(* IEC 61131-3 sources: generating_plc_code_with_llms/Code#2/ChatGPT_4/second run, 21 files *)

(* ---- 14.st ---- *)
// 34.95s
// 4
FUNCTION FC1001 : BOOL
VAR_INPUT
    MEW: REAL;  (* Measured value from the sensor *)
    SP: REAL;   (* Setpoint value *)
    HYS: REAL;  (* Hysteresis percentage *)
END_VAR
VAR_IN_OUT
    OUT: BOOL;  (* Output to be controlled *)
END_VAR
VAR
    P_HYS: REAL;  (* Absolute hysteresis value *)
END_VAR

P_HYS := SP * HYS / 100.0;  (* Calculate the hysteresis value *)

IF MEW > (SP + P_HYS) THEN
    OUT := TRUE;  (* Turn on output if measured value exceeds SP + hysteresis *)
ELSIF MEW < (SP - P_HYS) THEN
    OUT := FALSE;  (* Turn off output if measured value falls below SP - hysteresis *)
END_IF;

FC1001 := OUT;  (* Return the current state of the output *)

END_FUNCTION

(* ---- 15.st ---- *)
// 64.56s
// 4
FUNCTION FC1002 : BOOL
VAR_INPUT
    E_A : BOOL;     (* Switch for enabling/disabling the monitoring system *)
    SENSOR : BOOL;  (* Ultrasonic sensor input *)
    ZEITW : TIME;   (* Time duration for switching from warning to alarm *)
END_VAR
VAR_IN_OUT
    ZEIT : TON;     (* Timer for measuring the duration of perception *)
    P_HU : BOOL;    (* Horn for acoustic warning signal *)
    P_AL : BOOL;    (* Alarm signal *)
END_VAR

(* Monitoring system activation *)
IF E_A THEN
    (* When monitoring system is enabled *)
    IF SENSOR THEN
        ZEIT(IN := TRUE, PT := ZEITW);
        IF ZEIT.Q THEN
            P_HU := FALSE;  (* Turn off horn after time window *)
            P_AL := TRUE;   (* Activate alarm *)
        ELSE
            P_HU := TRUE;   (* Activate horn if object/person is detected *)
        END_IF;
    ELSE
        ZEIT(IN := FALSE);
        P_HU := FALSE;  (* Turn off horn if no object/person is detected *)
    END_IF;
ELSE
    (* When monitoring system is disabled *)
    P_HU := FALSE;
    P_AL := FALSE;
    ZEIT(IN := FALSE);
END_IF;

FC1002 := E_A;  (* Return the status of the monitoring system *)

END_FUNCTION

(* ---- 18.st ---- *)
// 37.69s
// 4
FUNCTION FC1003 : VOID
VAR_INPUT
    IN_R : REAL;      (* Input real value *)
    IN_MAX : REAL;    (* Input range maximum *)
    IN_MIN : REAL;    (* Input range minimum *)
    OUT_MAX : REAL;   (* Output range maximum *)
    OUT_MIN : REAL;   (* Output range minimum *)
END_VAR
VAR_OUTPUT
    OUT_R : REAL;     (* Output real value *)
    FEH : BOOL;       (* Error flag in case of invalid range *)
END_VAR
VAR_TEMP
    DIFF1 : REAL;     (* Temporary variable for differences *)
    DIFF2 : REAL;     (* Temporary variable for differences *)
END_VAR

(* Check for valid input range to avoid division by zero *)
IF IN_MAX <= IN_MIN THEN
    FEH := TRUE;
    RETURN;
END_IF;

(* Calculate the differences *)
DIFF1 := IN_MAX - IN_MIN;
DIFF2 := OUT_MAX - OUT_MIN;

(* Map the input value to the output range *)
OUT_R := OUT_MIN + ((IN_R - IN_MIN) * DIFF2) / DIFF1;

(* Set the error flag to false as no error occurred *)
FEH := FALSE;

END_FUNCTION

(* ---- 19.st ---- *)
// 43.16s
// 4
FUNCTION_BLOCK FB1005
VAR_INPUT
    START : BOOL;    (* Signal to start and end measurement *)
    DICKE : REAL;    (* Thickness measurement from lasers *)
    V_MAX : REAL;    (* Maximum tolerance value for thickness *)
    V_MIN : REAL;    (* Minimum tolerance value for thickness *)
END_VAR
VAR_OUTPUT
    D_MAX : REAL;    (* Maximum measured thickness *)
    D_MIN : REAL;    (* Minimum measured thickness *)
    P1 : BOOL;       (* Reject light indicator *)
END_VAR
VAR
    FO : BOOL;       (* Flag to indicate ongoing measurement *)
END_VAR

IF START THEN
    IF NOT FO THEN
        (* Start of a new measurement *)
        FO := TRUE;
        D_MAX := DICKE;
        D_MIN := DICKE;
    ELSE
        (* Ongoing measurement *)
        IF DICKE > D_MAX THEN
            D_MAX := DICKE;
        END_IF;

        IF DICKE < D_MIN THEN
            D_MIN := DICKE;
        END_IF;
    END_IF;
ELSE
    IF FO THEN
        (* End of measurement *)
        FO := FALSE;

        (* Check if measured values are outside tolerance range *)
        IF D_MAX > V_MAX OR D_MIN < V_MIN THEN
            P1 := TRUE;  (* Set reject light *)
        ELSE
            P1 := FALSE; (* Reset reject light *)
        END_IF;
    END_IF;
END_IF;

END_FUNCTION_BLOCK

(* ---- 20.st ---- *)
// 32.83s
// 3
FUNCTION_BLOCK INTERLOCK
VAR_INPUT
    I1 : BOOL;  (* Input for controlling Q1 *)
    I2 : BOOL;  (* Input for controlling Q2 *)
    TL : TIME;  (* Dead time between switching outputs *)
END_VAR
VAR_OUTPUT
    Q1 : BOOL;  (* Output Q1 *)
    Q2 : BOOL;  (* Output Q2 *)
END_VAR
VAR
    T1 : TOF;  (* Off-delay timer for Q1 *)
    T2 : TOF;  (* Off-delay timer for Q2 *)
END_VAR

(* Timer logic for Q1 *)
T1(IN := NOT Q1, PT := TL);
IF I1 AND T2.Q THEN
    Q1 := TRUE;
    Q2 := FALSE;
END_IF;

(* Timer logic for Q2 *)
T2(IN := NOT Q2, PT := TL);
IF I2 AND T1.Q THEN
    Q2 := TRUE;
    Q1 := FALSE;
END_IF;

END_FUNCTION_BLOCK

(* ---- 21.st ---- *)
// 144.85s
// weiter generieren
// 2
FUNCTION_BLOCK BURNER
VAR_INPUT
    IN : BOOL;
    STAGE2 : BOOL;
    OVER_TEMP : BOOL;
    OIL_TEMP : BOOL := TRUE;
    FLAME : BOOL;
    RST : BOOL;
    RST_TIMER : BOOL;
    PRE_HEAT_TIME : TIME := t#5s;
    PRE_VENT_TIME : TIME := t#15s;
    PRE_IGNITE_TIME : TIME := t#15s;
    POST_IGNITE_TIME : TIME := t#25s;
    STAGE2_DELAY : TIME := t#10s;
    SAFETY_TIME : TIME := t#5s;
    LOCKOUT_TIME : TIME := t#10s;
    MULTIPLE_IGNITION : BOOL := TRUE;
    KW1 : REAL;
    KW2 : REAL;
END_VAR
VAR_OUTPUT
    MOTOR : BOOL;
    COIL1 : BOOL;
    COIL2 : BOOL;
    PRE_HEAT : BOOL;
    IGNITE : BOOL;
    FAIL : BOOL;
    KWH : REAL;
    STATUS : BYTE;
END_VAR
VAR_IN_OUT
    RUNTIME1 : UDINT;
    RUNTIME2 : UDINT;
    CYCLES : UDINT;
END_VAR
VAR
    state : INT := 0;  (* Operational state of the burner *)
    last : TIME;  (* Last time an operation started *)
    tx : TIME;  (* Transition time for next state *)
    last_change : TIME;  (* Last time state changed *)
    timer1 : TON;  (* Timer for various operational delays *)
    timer2 : TON;  (* Timer for lockout period *)
    oil_temp_last : BOOL := FALSE;  (* Last state of OIL_TEMP *)
    cycles2 : UDINT;  (* Cycle count for stage 2 *)
END_VAR

(* Reset functionality *)
IF RST THEN
    state := 0;
    FAIL := FALSE;
    STATUS := 110;  (* Wait for Start signal *)
    timer2(IN := FALSE);  (* Reset lockout timer *)
    MOTOR := FALSE;
    PRE_HEAT := FALSE;
    IGNITE := FALSE;
    COIL1 := FALSE;
    COIL2 := FALSE;
    RETURN;
END_IF;

(* Lockout timer check *)
timer2(IN := RST_TIMER, PT := LOCKOUT_TIME);
IF timer2.Q THEN
    RST_TIMER := FALSE;  (* Reset RST_TIMER after lockout period *)
END_IF;

(* Main state machine for burner operation *)
CASE state OF
    0:
        IF IN AND NOT OVER_TEMP AND NOT timer2.Q THEN
            state := 1;
            PRE_HEAT := TRUE;
            last_change := tx;
            timer1(IN := TRUE, PT := PRE_HEAT_TIME);
        END_IF;
    1:
        IF timer1.Q THEN
            IF NOT OIL_TEMP THEN
                FAIL := TRUE;
                STATUS := 1;  (* Fuel oil warming has not responded within PRE_HEAT_TIME *)
                state := 9;  (* Error state *)
            ELSE
                state := 2;  (* Proceed to next stage *)
                MOTOR := TRUE;
                last_change := tx;
                timer1(IN := TRUE, PT := PRE_VENT_TIME);  (* Start ventilation period *)
            END_IF;
        END_IF;
    2:
        IF timer1.Q THEN
            state := 3;
            IGNITE := TRUE;
            last_change := tx;
            timer1(IN := TRUE, PT := PRE_IGNITE_TIME + SAFETY_TIME);  (* Ignition and safety period *)
        END_IF;
    3:
        IF FLAME THEN
            state := 4;
            COIL1 := TRUE;  (* Burner running on stage 1 *)
            STATUS := 112;
            last_change := tx;
            RUNTIME1 := RUNTIME1 + 1;
            IF STAGE2 THEN
                timer1(IN := TRUE, PT := STAGE2_DELAY);  (* Delay for stage 2 activation *)
            END_IF;
        ELSIF timer1.Q THEN
            FAIL := TRUE;
            STATUS := 4;  (* Safety time was passed without a flame *)
            state := 9;  (* Error state *)
        END_IF;
    4:
        IF timer1.Q AND STAGE2 THEN
            state := 5;
            COIL2 := TRUE;  (* Burner running on stage 2 *)
            STATUS := 113;
            RUNTIME2 := RUNTIME2 + 1;
        END_IF;
    9:
        MOTOR := FALSE;
        PRE_HEAT := FALSE;
        IGNITE := FALSE;
        COIL1 := FALSE;
        COIL2 := FALSE;
        RST_TIMER := TRUE;  (* Start lockout timer *)
        state := 0;  (* Reset state after handling error *)
END_CASE;

(* Handle OVER_TEMP condition *)
IF OVER_TEMP THEN
    FAIL := TRUE;
    STATUS := 9;  (* Boiler overheating contact has tripped *)
    MOTOR := FALSE;
    PRE_HEAT := FALSE;
    IGNITE := FALSE;
    COIL1 := FALSE;
    COIL2 := FALSE;
    state := 9;  (* Set error state *)
END_IF;

END_FUNCTION_BLOCK

(* ---- 1.st ---- *)
// 18.4s
// 4
VAR
    xAllOn : BOOL;
    xAllOff : BOOL;
    xAlarm1 : BOOL;
    xAlarm2 : BOOL;
END_VAR

IF xAllOn THEN
    xAlarm1 := TRUE;
    xAlarm2 := TRUE;
    xAllOn := FALSE;
END_IF;

IF xAllOff THEN
    xAlarm1 := FALSE;
    xAlarm2 := FALSE;
    xAllOff := FALSE;
END_IF;

(* ---- 10.st ---- *)
// 16.0s
// 4
VAR_INPUT
    X : REAL;
END_VAR

VAR
    SigmoidResult : REAL;
END_VAR

SigmoidResult := 1 / (1 + EXP(-X));

(* ---- 11.st ---- *)
// 17.44s
// 4
VAR_INPUT
    x : REAL;  (* Input number *)
END_VAR

VAR
    signResult : INT;  (* Result of the sign function *)
END_VAR

IF x > 0 THEN
    signResult := 1;  (* Positive number *)
ELSIF x < 0 THEN
    signResult := -1;  (* Negative number *)
ELSE
    signResult := 0;  (* Zero *)
END_IF;

(* ---- 12.st ---- *)
// 13.41s
// 4
VAR
    X : REAL;         (* Input for the hyperbolic sine function *)
    SinhResult : REAL; (* Result of sinh(x) *)
END_VAR

SinhResult := (EXP(X) - EXP(-X)) / 2;

(* ---- 13.st ---- *)
// 20.21s
// 2
VAR CONSTANT
    MAXNUMBERS : UINT := 99;  (* The upper index of the array *)
END_VAR

VAR
    aNumbers : ARRAY[0..MAXNUMBERS] OF INT;  (* Array of 100 random numbers *)
    nCnt : INT;                              (* Counter for the loop *)
END_VAR

nCnt := 0;

REPEAT
    IF aNumbers[nCnt] = 10 THEN
        EXIT;  (* Exit the loop if the number 10 is found *)
    END_IF;

    nCnt := nCnt + 1;
UNTIL nCnt > MAXNUMBERS;  (* Continue until the end of the array is reached *)

(* ---- 16.st ---- *)
// 57.71s
// 4
VAR
    North_green : BOOL;
    North_yellow : BOOL;
    North_red : BOOL;
    East_green : BOOL;
    East_yellow : BOOL;
    East_red : BOOL;
    T1 : TON;
END_VAR

(* Start the timer *)
T1(IN := TRUE, PT := T#10000MS);

(* Control the North and East traffic lights based on the elapsed time of the timer *)
IF T1.ET < T#5000MS THEN
    (* 0ms to 5000ms: North green, East red *)
    North_green := TRUE;
    North_yellow := FALSE;
    North_red := FALSE;
    East_green := FALSE;
    East_yellow := FALSE;
    East_red := TRUE;
ELSIF T1.ET < T#5500MS THEN
    (* 5000ms to 5500ms: North yellow, East red *)
    North_green := FALSE;
    North_yellow := TRUE;
    North_red := FALSE;
    East_green := FALSE;
    East_yellow := FALSE;
    East_red := TRUE;
ELSIF T1.ET < T#9500MS THEN
    (* 5500ms to 9500ms: North red, East green *)
    North_green := FALSE;
    North_yellow := FALSE;
    North_red := TRUE;
    East_green := TRUE;
    East_yellow := FALSE;
    East_red := FALSE;
ELSE
    (* 9500ms to 10000ms: North red, East yellow *)
    North_green := FALSE;
    North_yellow := FALSE;
    North_red := TRUE;
    East_green := FALSE;
    East_yellow := TRUE;
    East_red := FALSE;
END_IF;

(* Reset the timer at the end of the cycle *)
IF T1.Q THEN
    T1.IN := FALSE;
    T1(IN := TRUE);  (* Restart the timer *)
END_IF;

(* ---- 17.st ---- *)
// 28.0s
// 3
VAR
    aiOutside : INT;       (* Analog input for outside temperature *)
    aiHumidity : INT;      (* Analog input for humidity *)
    sShowText : STRING[80];(* String to display the message *)
END_VAR

(* Convert the analog inputs to temperature and humidity values *)
(* Assuming the range of the analog input is from 0 to 32767 and this corresponds to -40 to 60 °C for temperature and 0 to 100% for humidity *)
VAR
    fTemperature : REAL; (* Temperature in degrees Celsius *)
    fHumidity : REAL;    (* Humidity in percentage *)
END_VAR

fTemperature := (aiOutside / 32767.0) * 100.0 - 40.0;  (* Conversion formula *)
fHumidity := (aiHumidity / 32767.0) * 100.0;           (* Conversion formula *)

(* Evaluate temperature and humidity to set the display text *)
IF fTemperature < 18 THEN
    sShowText := 'Cold';
ELSIF fTemperature <= 25 THEN
    IF fHumidity >= 40 AND fHumidity <= 75 THEN
        sShowText := 'Opt';
    ELSE
        sShowText := 'Temp. OK';
    END_IF;
ELSE
    sShowText := 'Hot';
END_IF;

(* ---- 2.st ---- *)
// 26.75s
// 4
VAR_INPUT
    N : INT;
    K : INT;
END_VAR

VAR
    Result : LREAL;  (* Using LREAL for potentially large results *)
    i : INT;
END_VAR

(* Initialize result *)
Result := 1;

(* Adjust K for optimization *)
IF K > N - K THEN
    K := N - K;
END_IF;

(* Calculate binomial coefficient *)
FOR i := 0 TO K - 1 DO
    Result := Result * (N - i) / (i + 1);
END_FOR;

(* ---- 3.st ---- *)
// 17.02s
// 3
VAR_INPUT
    X : INT;
END_VAR

VAR
    t1 : DINT := 0;
    t2 : DINT := 1;
    nextTerm : DINT := 0;
    i : INT;
END_VAR

IF X = 0 THEN
    nextTerm := 0;
ELSIF X = 1 THEN
    nextTerm := 1;
ELSE
    FOR i := 2 TO X DO
        nextTerm := t1 + t2;
        t1 := t2;
        t2 := nextTerm;
    END_FOR;
END_IF;

(* ---- 4.st ---- *)
// 26.41s
// 2
VAR
    aiLevel : INT;           (* Analog input representing the fill level *)
    PercentLevel : UINT;     (* Fill level as a percentage *)
    doLow : BOOL;            (* Output for low level indication *)
    doOk : BOOL;             (* Output for ok level indication *)
    doHigh : BOOL;           (* Output for high level indication *)
    doAlarm : BOOL;          (* Output for alarm indication *)
END_VAR

(* Convert the analog input to a percentage *)
PercentLevel := UINT(aiLevel * 100 / 32767);

(* Check the level and set outputs accordingly *)
CASE PercentLevel OF
    0..1:
        BEGIN
            doLow := TRUE;
            doOk := FALSE;
            doHigh := FALSE;
            doAlarm := TRUE; (* Activate alarm for less than 1% *)
        END
    2..79:
        BEGIN
            doLow := FALSE;
            doOk := TRUE;
            doHigh := FALSE;
            doAlarm := FALSE;
        END
    80..100:
        BEGIN
            doLow := FALSE;
            doOk := FALSE;
            doHigh := TRUE;
            doAlarm := FALSE;
        END
END_CASE;

(* ---- 5.st ---- *)
// 50.7s
// 4
VAR
    Start_Loop : BOOL := FALSE;
    one_hour : TIME := T#1h;            (* 1 hour duration for timer *)
    One_Hour_Timer : TON;               (* Timer for 1 hour countdown *)
    Gate_Open : BOOL := FALSE;          (* Indicates if gate is open *)
    Close_Gate_Inst : BOOL := FALSE;    (* Instruction to close gate *)
    Sensed_Car : BOOL := FALSE;         (* Detects presence of car *)
    Sensed_Car_Inst : BOOL := FALSE;    (* Car detection instance *)
    Sensed_App : BOOL := FALSE;         (* Detects signal from app *)
    Mobile_Inst : BOOL := FALSE;        (* Mobile app detection instance *)
    Auth : STRING;                      (* Authentication string *)
    my_defined_str : STRING := 'abcd';  (* Defined authentication string *)
END_VAR

(* Timer control *)
IF Start_Loop = FALSE THEN
    One_Hour_Timer(IN := TRUE, PT := one_hour);
ELSE
    One_Hour_Timer(IN := FALSE);
END_IF;

(* Check if timer has timed out and gate is open *)
IF One_Hour_Timer.Q AND Gate_Open THEN
    Close_Gate_Inst := TRUE;
    Gate_Open := FALSE;
END_IF;

(* Check for car or app presence and correct authentication *)
IF (Sensed_Car OR Sensed_App) AND (Auth = my_defined_str) THEN
    Gate_Open := TRUE;
    Sensed_Car_Inst := Sensed_Car;
    Mobile_Inst := Sensed_App;
ELSE
    IF NOT One_Hour_Timer.Q THEN
        Close_Gate_Inst := FALSE;
    END_IF;
END_IF;

(* ---- 6.st ---- *)
// 47.53s
// 3
VAR CONSTANT
    WAIT : UINT := 0;
    TOP_POSITION : UINT := 1;
    BOTTOM_POSITION : UINT := 2;
    GETBOX : UINT := 3;
    UNLOAD_POSITION : UINT := 4;
    UNLOAD_BOX : UINT := 5;
END_VAR

VAR
    (* digital outputs *)
    doConvTop : BOOL;
    doConvBottom : BOOL;
    doConvLift : BOOL;
    doLiftTop : BOOL;
    doLiftBottom : BOOL;
    doLiftUnload : BOOL;
    (* digital inputs *)
    diConvTop : BOOL;
    diConvBottom : BOOL;
    diLiftTop : BOOL;
    diLiftBottom : BOOL;
    diLiftUnload : BOOL;
    diBoxLift : BOOL;
    (* status variables *)
    selectLift : UINT;
    ConvTopOn : BOOL;
    ConvBottomOn : BOOL;
END_VAR

(* Handle the conveyor belts *)
IF diConvTop THEN
    doConvTop := FALSE;
    selectLift := TOP_POSITION;
END_IF;

IF diConvBottom THEN
    doConvBottom := FALSE;
    selectLift := BOTTOM_POSITION;
END_IF;

(* Control the lift *)
CASE selectLift OF
    TOP_POSITION:
        IF NOT diLiftTop THEN
            doLiftTop := TRUE;
            doLiftBottom := FALSE;
            doLiftUnload := FALSE;
        ELSIF diLiftTop THEN
            doConvLift := TRUE;
            IF diBoxLift THEN
                selectLift := UNLOAD_POSITION;
            END_IF;
        END_IF;

    BOTTOM_POSITION:
        IF NOT diLiftBottom THEN
            doLiftBottom := TRUE;
            doLiftTop := FALSE;
            doLiftUnload := FALSE;
        ELSIF diLiftBottom THEN
            doConvLift := TRUE;
            IF diBoxLift THEN
                selectLift := UNLOAD_POSITION;
            END_IF;
        END_IF;

    UNLOAD_POSITION:
        doConvLift := FALSE;
        doLiftUnload := TRUE;
        IF diLiftUnload THEN
            selectLift := UNLOAD_BOX;
        END_IF;

    UNLOAD_BOX:
        doLiftUnload := FALSE;
        IF NOT diBoxLift THEN
            selectLift := WAIT;
        END_IF;

    WAIT:
        doLiftTop := FALSE;
        doLiftBottom := FALSE;
        doLiftUnload := FALSE;
END_CASE;

(* ---- 7.st ---- *)
// 18.24s
// 2
VAR CONSTANT
    MAX_INDEX: USINT := 4;  (* Represents the highest index for load receptors *)
END_VAR

VAR
    aWeights : ARRAY[0..MAX_INDEX] OF INT;  (* Array of load values from receptors *)
    iCnt : USINT;                           (* Loop counter *)
    sumWeight : DINT;                       (* Total sum of weights *)
    avgWeight : INT;                        (* Average weight *)
END_VAR

(* Initialize sum *)
sumWeight := 0;

(* Calculate the sum of the weights *)
FOR iCnt := 0 TO MAX_INDEX DO
    sumWeight := sumWeight + aWeights[iCnt];
END_FOR;

(* Calculate the average weight, dividing by the number of receptors *)
avgWeight := sumWeight / (MAX_INDEX + 1);

(* ---- 8.st ---- *)
// 29.25s
// 3
VAR_INPUT
    X : REAL;  (* Input for the Lambert W function *)
END_VAR

VAR
    w : REAL;      (* Approximation of W(x) *)
    i : INT;       (* Iteration counter *)
    we : REAL;     (* w * exp(w) *)
    w1e : REAL;    (* (w + 1) * exp(w) *)
    ewx : REAL;    (* exp(w) - X/w *)
    last : DWORD;  (* To check for convergence *)
END_VAR

(* Initial guess *)
IF X = 0 THEN
    w := 0;
ELSE
    w := LOG(X);  (* Logarithmic approximation for starting value *)
END_IF;

last := TO_DWORD(w);
FOR i := 1 TO 100 DO  (* Limiting iterations to 100 for safety *)
    we := w * EXP(w);
    w1e := (w + 1) * EXP(w);
    ewx := EXP(w) - X / w;

    (* Newton's Method update *)
    w := w - we / (w1e - ewx);

    (* Check for convergence *)
    IF last = TO_DWORD(w) THEN
        EXIT;  (* Exit loop if converged *)
    END_IF;
    last := TO_DWORD(w);
END_FOR;

(* ---- 9.st ---- *)
// 18.49s
// 4
VAR
    YEAR : INT;
    IsLeapYear : BOOL;
END_VAR

IsLeapYear := FALSE;  (* Default assumption *)

IF (YEAR MOD 4 = 0) THEN
    IF (YEAR MOD 100 = 0) THEN
        IF (YEAR MOD 400 = 0) THEN
            IsLeapYear := TRUE;  (* Divisible by 400, so it's a leap year *)
        END_IF;
    ELSE
        IsLeapYear := TRUE;  (* Divisible by 4 but not by 100, so it's a leap year *)
    END_IF;
END_IF;
